// TIA Portal project "babu_singlePushButtonWorking" (V15)

(* hardware
DEVICE "S7-1200 station_1"  S7-1200 Station
   slot 0: "Rack_0"  S7-1200 Rack  Rack  V1.0
   slot 1: "PLC_1"  CPU 1212C DC/DC/DC  6ES7 212-1AE40-0XB0  V4.2
*)

// ===== PLC "PLC_1"  CPU 1212C DC/DC/DC =====

VAR_GLOBAL   // PLC tag table "Default tag table"
   "PUSH BUTTON" AT %M0.0 : Bool;
   "MEMORY 1" AT %M0.1 : Bool;
   "MEMORY 2" AT %M0.2 : Bool;
   "MEMORY 3" AT %M0.3 : Bool;
   "BULB" AT %Q0.0 : Bool;
END_VAR

ORGANIZATION_BLOCK "Main"   // OB1, LAD, ProgramCycle
TITLE = "Main Program Sweep (Cycle)"
{ S7_Optimized_Access := 'TRUE' }
VERSION : 0.1
   VAR_INPUT
      Initial_Call : Bool;   // Initial call of this OB
      Remanence : Bool;   // =True, if remanent data are available
   END_VAR
BEGIN

REGION Network 1
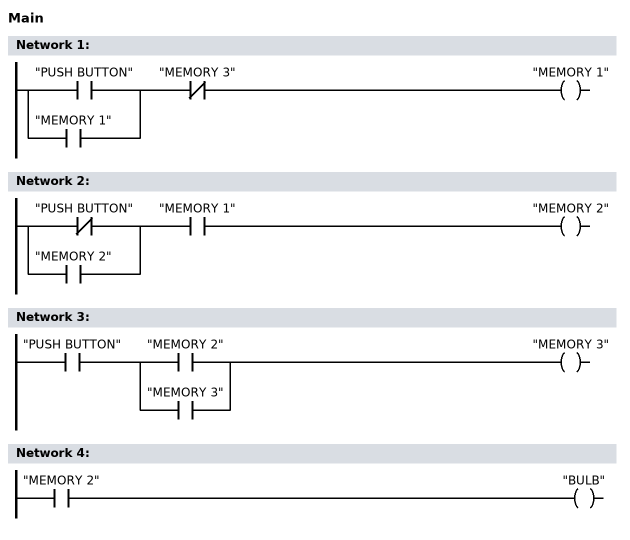
   RUNG wire#powerrail
      Contact( "PUSH BUTTON" )
      wire#w1
      I_Contact( "MEMORY 3" )
      Coil( "MEMORY 1" )
   END_RUNG
   RUNG wire#powerrail
      Contact( "MEMORY 1" )
   END_RUNG wire#w1
   // the same network as SCL:
   "MEMORY 1" := ("PUSH BUTTON" OR "MEMORY 1") AND NOT "MEMORY 3";
END_REGION

REGION Network 2
   RUNG wire#powerrail
      I_Contact( "PUSH BUTTON" )
      wire#w1
      Contact( "MEMORY 1" )
      Coil( "MEMORY 2" )
   END_RUNG
   RUNG wire#powerrail
      Contact( "MEMORY 2" )
   END_RUNG wire#w1
   // the same network as SCL:
   "MEMORY 2" := (NOT "PUSH BUTTON" OR "MEMORY 2") AND "MEMORY 1";
END_REGION

REGION Network 3
   RUNG wire#powerrail
      Contact( "PUSH BUTTON" )
      wire#w1
      Contact( "MEMORY 2" )
      wire#w2
      Coil( "MEMORY 3" )
   END_RUNG
   RUNG wire#w1
      Contact( "MEMORY 3" )
   END_RUNG wire#w2
   // the same network as SCL:
   "MEMORY 3" := "PUSH BUTTON" AND ("MEMORY 2" OR "MEMORY 3");
END_REGION

REGION Network 4
   RUNG wire#powerrail
      Contact( "MEMORY 2" )
      Coil( "BULB" )
   END_RUNG
   // the same network as SCL:
   "BULB" := "MEMORY 2";
END_REGION
END_ORGANIZATION_BLOCK